Staubli VAL3: test_com.pgx

program test_com()
begin
  while true
    doECAT1_0 = true

    if(diECAT1_0 == true)

      doECAT1_0 = false

      open(tTool)
      movej(jP1, tTool, mNomSpeed)
      movej(jP2, tTool, mNomSpeed)
      close(tTool)
      movej(jP4, tTool, mNomSpeed)
      movej(jP5, tTool, mNomSpeed)
      movej(jP3, tTool, mNomSpeed)
      open(tTool)
      movej(jP1, tTool, mNomSpeed)
      movej(jP3, tTool, mNomSpeed)
      close(tTool)
      movej(jP5, tTool, mNomSpeed)
      movej(jP4, tTool, mNomSpeed)
      movej(jP2, tTool, mNomSpeed)
      open(tTool)
      waitEndMove()

      doECAT1_0 = true

    endIf
  endWhile
end
